// Mitsubishi GX Works2 project: Q-123_E_MTL   PLC: Q06H
// MDAS sample program

PROGRAM Q  // MDAS
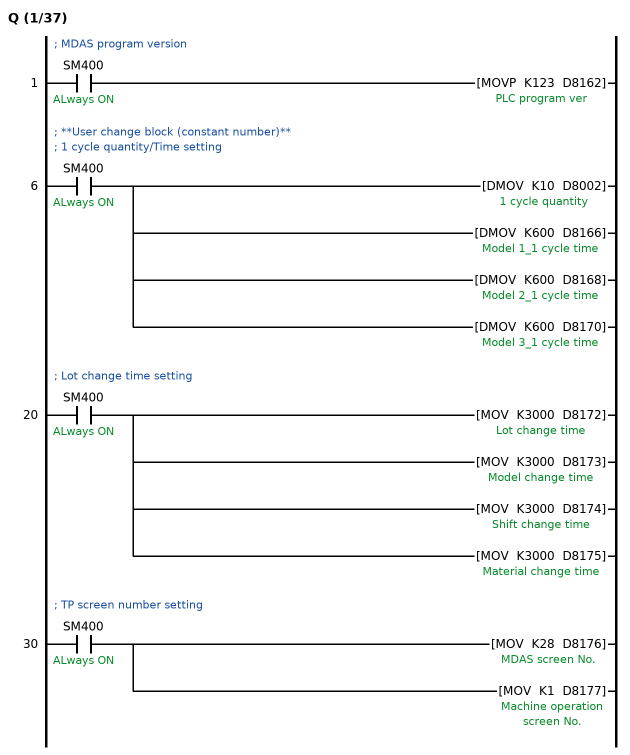
; MDAS program version
1     LD      SM400  ; ALways ON
      MOVP    K123 D8162  ; PLC program ver
; **User change block (constant number)**
; 1 cycle quantity/Time setting
6     LD      SM400  ; ALways ON
      DMOV    K10 D8002  ; 1 cycle quantity
      DMOV    K600 D8166  ; Model 1_1 cycle time
      DMOV    K600 D8168  ; Model 2_1 cycle time
      DMOV    K600 D8170  ; Model 3_1 cycle time
; Lot change time setting
20    LD      SM400  ; ALways ON
      MOV     K3000 D8172  ; Lot change time
      MOV     K3000 D8173  ; Model change time
      MOV     K3000 D8174  ; Shift change time
      MOV     K3000 D8175  ; Material change time
; TP screen number setting
30    LD      SM400  ; ALways ON
      MOV     K28 D8176  ; MDAS screen No.
      MOV     K1 D8177  ; Machine operation screen No.
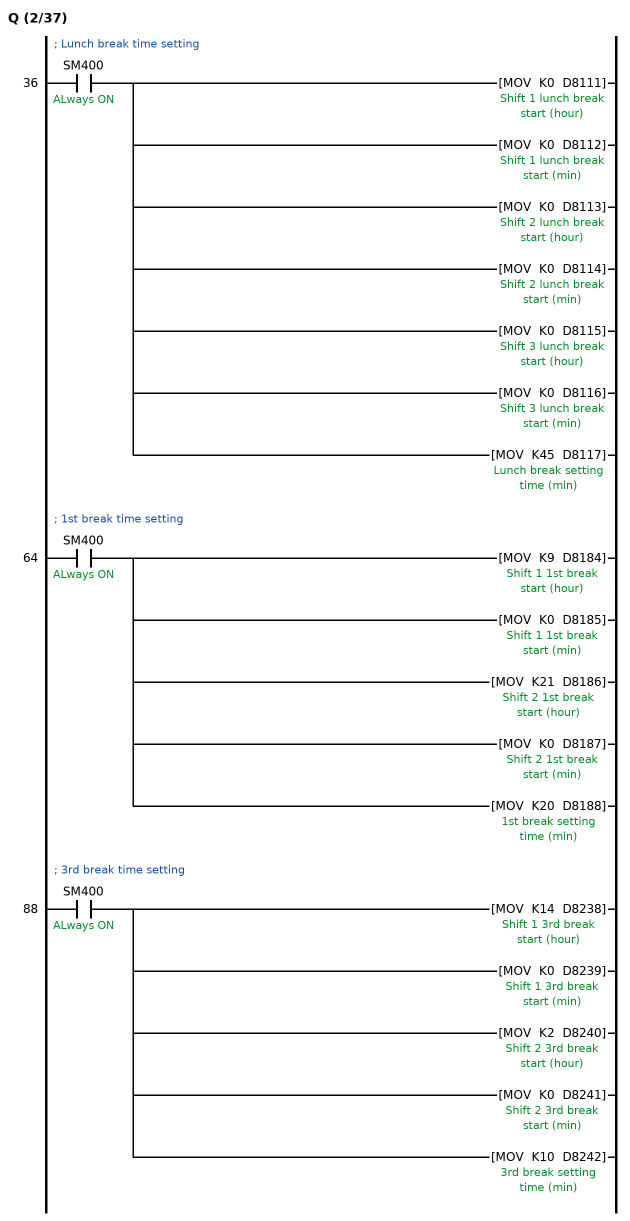
; Lunch break time setting
36    LD      SM400  ; ALways ON
      MOV     K0 D8111  ; Shift 1 lunch break start (hour)
      MOV     K0 D8112  ; Shift 1 lunch break start (min)
      MOV     K0 D8113  ; Shift 2 lunch break start (hour)
      MOV     K0 D8114  ; Shift 2 lunch break start (min)
      MOV     K0 D8115  ; Shift 3 lunch break start (hour)
      MOV     K0 D8116  ; Shift 3 lunch break start (min)
      MOV     K45 D8117  ; Lunch break setting time (min)
; 1st break time setting
64    LD      SM400  ; ALways ON
      MOV     K9 D8184  ; Shift 1 1st break start (hour)
      MOV     K0 D8185  ; Shift 1 1st break start (min)
      MOV     K21 D8186  ; Shift 2 1st break start (hour)
      MOV     K0 D8187  ; Shift 2 1st break start (min)
      MOV     K20 D8188  ; 1st break setting time (min)
; 3rd break time setting
88    LD      SM400  ; ALways ON
      MOV     K14 D8238  ; Shift 1 3rd break start (hour)
      MOV     K0 D8239  ; Shift 1 3rd break start (min)
      MOV     K2 D8240  ; Shift 2 3rd break start (hour)
      MOV     K0 D8241  ; Shift 2 3rd break start (min)
      MOV     K10 D8242  ; 3rd break setting time (min)
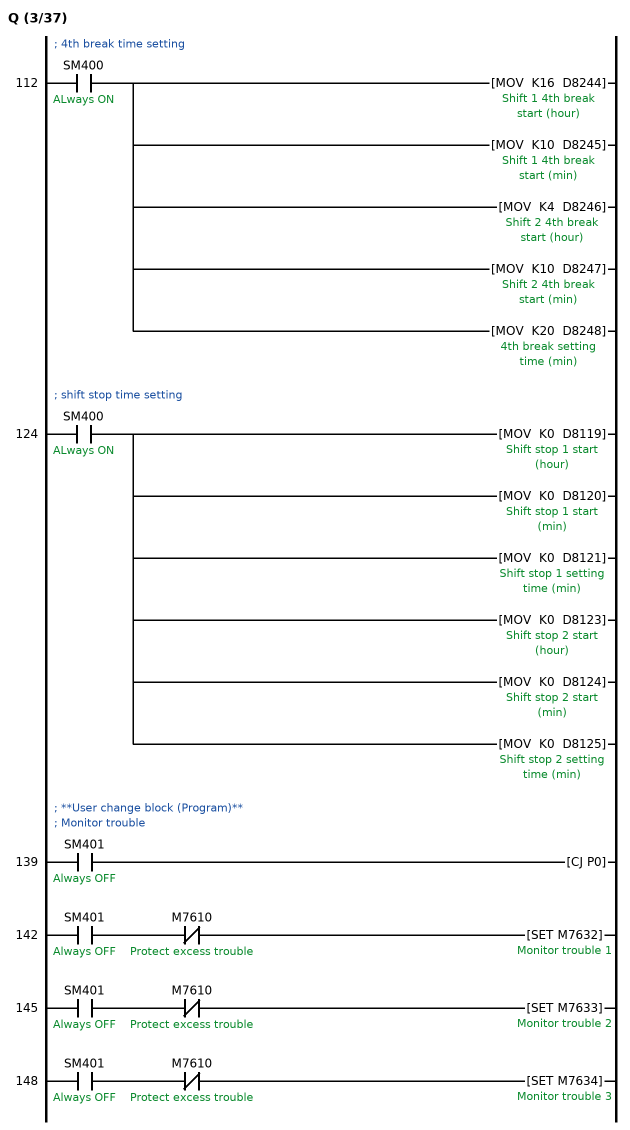
; 4th break time setting
112   LD      SM400  ; ALways ON
      MOV     K16 D8244  ; Shift 1 4th break start (hour)
      MOV     K10 D8245  ; Shift 1 4th break start (min)
      MOV     K4 D8246  ; Shift 2 4th break start (hour)
      MOV     K10 D8247  ; Shift 2 4th break start (min)
      MOV     K20 D8248  ; 4th break setting time (min)
; shift stop time setting
124   LD      SM400  ; ALways ON
      MOV     K0 D8119  ; Shift stop 1 start (hour)
      MOV     K0 D8120  ; Shift stop 1 start (min)
      MOV     K0 D8121  ; Shift stop 1 setting time (min)
      MOV     K0 D8123  ; Shift stop 2 start (hour)
      MOV     K0 D8124  ; Shift stop 2 start (min)
      MOV     K0 D8125  ; Shift stop 2 setting time (min)
; **User change block (Program)**
; Monitor trouble
139   LD      SM401  ; Always OFF
      CJ      P0
142   LD      SM401  ; Always OFF
      ANI     M7610  ; Protect excess trouble
      SET     M7632  ; Monitor trouble 1
145   LD      SM401  ; Always OFF
      ANI     M7610  ; Protect excess trouble
      SET     M7633  ; Monitor trouble 2
148   LD      SM401  ; Always OFF
      ANI     M7610  ; Protect excess trouble
      SET     M7634  ; Monitor trouble 3
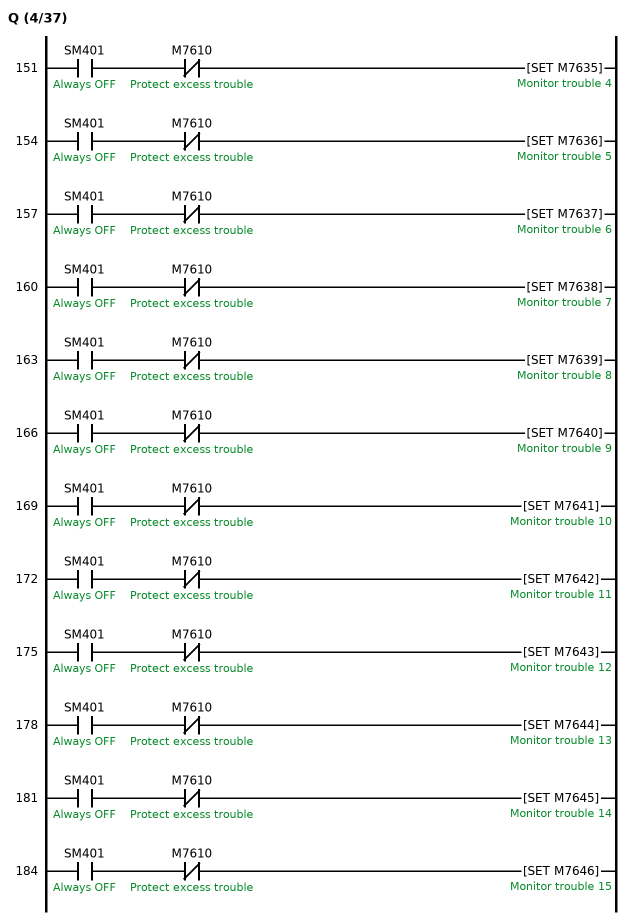
151   LD      SM401  ; Always OFF
      ANI     M7610  ; Protect excess trouble
      SET     M7635  ; Monitor trouble 4
154   LD      SM401  ; Always OFF
      ANI     M7610  ; Protect excess trouble
      SET     M7636  ; Monitor trouble 5
157   LD      SM401  ; Always OFF
      ANI     M7610  ; Protect excess trouble
      SET     M7637  ; Monitor trouble 6
160   LD      SM401  ; Always OFF
      ANI     M7610  ; Protect excess trouble
      SET     M7638  ; Monitor trouble 7
163   LD      SM401  ; Always OFF
      ANI     M7610  ; Protect excess trouble
      SET     M7639  ; Monitor trouble 8
166   LD      SM401  ; Always OFF
      ANI     M7610  ; Protect excess trouble
      SET     M7640  ; Monitor trouble 9
169   LD      SM401  ; Always OFF
      ANI     M7610  ; Protect excess trouble
      SET     M7641  ; Monitor trouble 10
172   LD      SM401  ; Always OFF
      ANI     M7610  ; Protect excess trouble
      SET     M7642  ; Monitor trouble 11
175   LD      SM401  ; Always OFF
      ANI     M7610  ; Protect excess trouble
      SET     M7643  ; Monitor trouble 12
178   LD      SM401  ; Always OFF
      ANI     M7610  ; Protect excess trouble
      SET     M7644  ; Monitor trouble 13
181   LD      SM401  ; Always OFF
      ANI     M7610  ; Protect excess trouble
      SET     M7645  ; Monitor trouble 14
184   LD      SM401  ; Always OFF
      ANI     M7610  ; Protect excess trouble
      SET     M7646  ; Monitor trouble 15
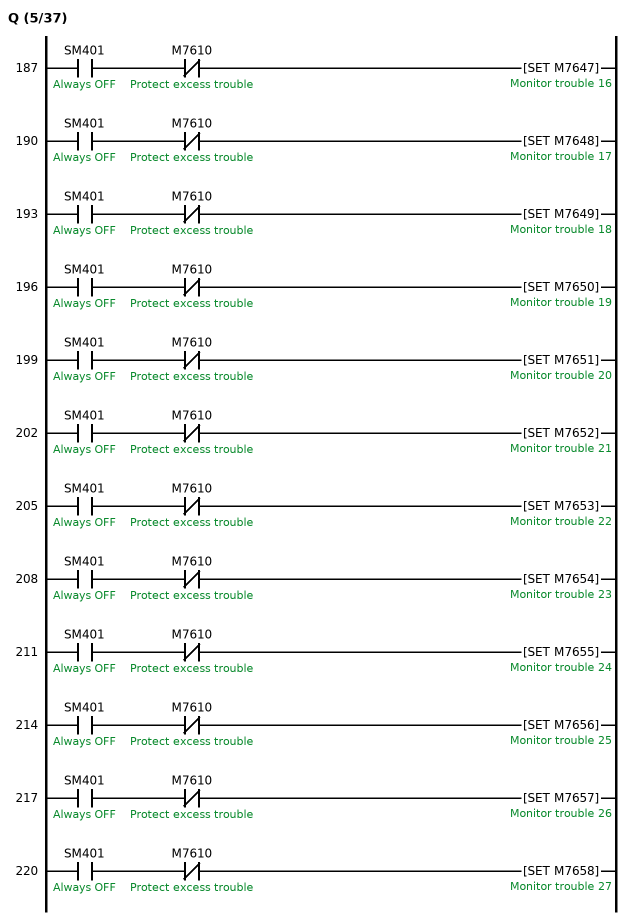
187   LD      SM401  ; Always OFF
      ANI     M7610  ; Protect excess trouble
      SET     M7647  ; Monitor trouble 16
190   LD      SM401  ; Always OFF
      ANI     M7610  ; Protect excess trouble
      SET     M7648  ; Monitor trouble 17
193   LD      SM401  ; Always OFF
      ANI     M7610  ; Protect excess trouble
      SET     M7649  ; Monitor trouble 18
196   LD      SM401  ; Always OFF
      ANI     M7610  ; Protect excess trouble
      SET     M7650  ; Monitor trouble 19
199   LD      SM401  ; Always OFF
      ANI     M7610  ; Protect excess trouble
      SET     M7651  ; Monitor trouble 20
202   LD      SM401  ; Always OFF
      ANI     M7610  ; Protect excess trouble
      SET     M7652  ; Monitor trouble 21
205   LD      SM401  ; Always OFF
      ANI     M7610  ; Protect excess trouble
      SET     M7653  ; Monitor trouble 22
208   LD      SM401  ; Always OFF
      ANI     M7610  ; Protect excess trouble
      SET     M7654  ; Monitor trouble 23
211   LD      SM401  ; Always OFF
      ANI     M7610  ; Protect excess trouble
      SET     M7655  ; Monitor trouble 24
214   LD      SM401  ; Always OFF
      ANI     M7610  ; Protect excess trouble
      SET     M7656  ; Monitor trouble 25
217   LD      SM401  ; Always OFF
      ANI     M7610  ; Protect excess trouble
      SET     M7657  ; Monitor trouble 26
220   LD      SM401  ; Always OFF
      ANI     M7610  ; Protect excess trouble
      SET     M7658  ; Monitor trouble 27
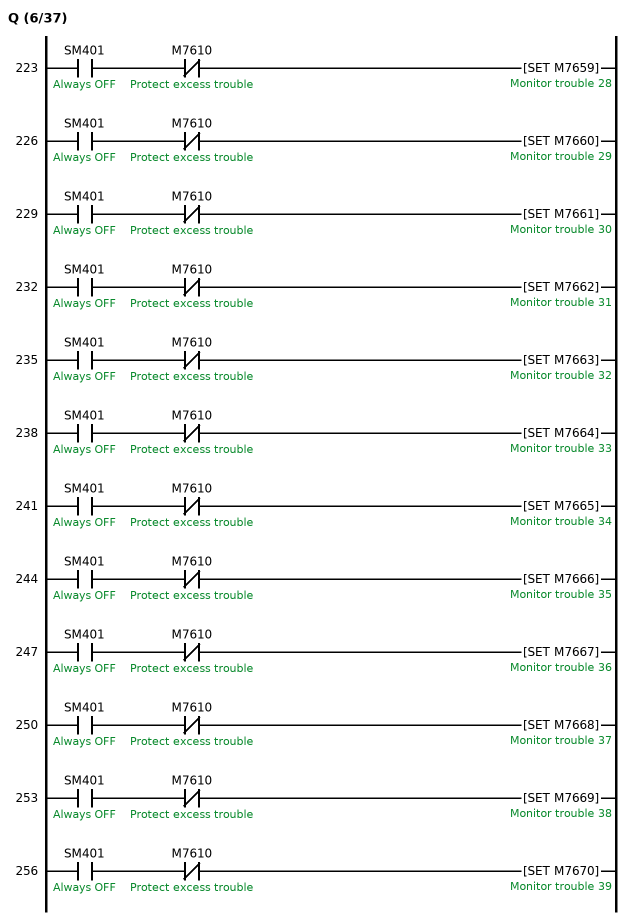
223   LD      SM401  ; Always OFF
      ANI     M7610  ; Protect excess trouble
      SET     M7659  ; Monitor trouble 28
226   LD      SM401  ; Always OFF
      ANI     M7610  ; Protect excess trouble
      SET     M7660  ; Monitor trouble 29
229   LD      SM401  ; Always OFF
      ANI     M7610  ; Protect excess trouble
      SET     M7661  ; Monitor trouble 30
232   LD      SM401  ; Always OFF
      ANI     M7610  ; Protect excess trouble
      SET     M7662  ; Monitor trouble 31
235   LD      SM401  ; Always OFF
      ANI     M7610  ; Protect excess trouble
      SET     M7663  ; Monitor trouble 32
238   LD      SM401  ; Always OFF
      ANI     M7610  ; Protect excess trouble
      SET     M7664  ; Monitor trouble 33
241   LD      SM401  ; Always OFF
      ANI     M7610  ; Protect excess trouble
      SET     M7665  ; Monitor trouble 34
244   LD      SM401  ; Always OFF
      ANI     M7610  ; Protect excess trouble
      SET     M7666  ; Monitor trouble 35
247   LD      SM401  ; Always OFF
      ANI     M7610  ; Protect excess trouble
      SET     M7667  ; Monitor trouble 36
250   LD      SM401  ; Always OFF
      ANI     M7610  ; Protect excess trouble
      SET     M7668  ; Monitor trouble 37
253   LD      SM401  ; Always OFF
      ANI     M7610  ; Protect excess trouble
      SET     M7669  ; Monitor trouble 38
256   LD      SM401  ; Always OFF
      ANI     M7610  ; Protect excess trouble
      SET     M7670  ; Monitor trouble 39
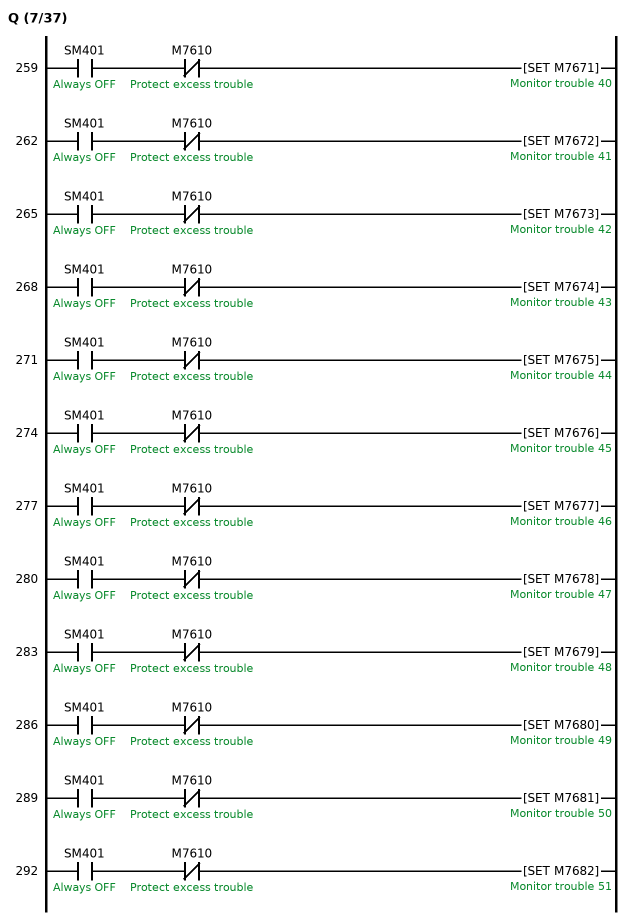
259   LD      SM401  ; Always OFF
      ANI     M7610  ; Protect excess trouble
      SET     M7671  ; Monitor trouble 40
262   LD      SM401  ; Always OFF
      ANI     M7610  ; Protect excess trouble
      SET     M7672  ; Monitor trouble 41
265   LD      SM401  ; Always OFF
      ANI     M7610  ; Protect excess trouble
      SET     M7673  ; Monitor trouble 42
268   LD      SM401  ; Always OFF
      ANI     M7610  ; Protect excess trouble
      SET     M7674  ; Monitor trouble 43
271   LD      SM401  ; Always OFF
      ANI     M7610  ; Protect excess trouble
      SET     M7675  ; Monitor trouble 44
274   LD      SM401  ; Always OFF
      ANI     M7610  ; Protect excess trouble
      SET     M7676  ; Monitor trouble 45
277   LD      SM401  ; Always OFF
      ANI     M7610  ; Protect excess trouble
      SET     M7677  ; Monitor trouble 46
280   LD      SM401  ; Always OFF
      ANI     M7610  ; Protect excess trouble
      SET     M7678  ; Monitor trouble 47
283   LD      SM401  ; Always OFF
      ANI     M7610  ; Protect excess trouble
      SET     M7679  ; Monitor trouble 48
286   LD      SM401  ; Always OFF
      ANI     M7610  ; Protect excess trouble
      SET     M7680  ; Monitor trouble 49
289   LD      SM401  ; Always OFF
      ANI     M7610  ; Protect excess trouble
      SET     M7681  ; Monitor trouble 50
292   LD      SM401  ; Always OFF
      ANI     M7610  ; Protect excess trouble
      SET     M7682  ; Monitor trouble 51
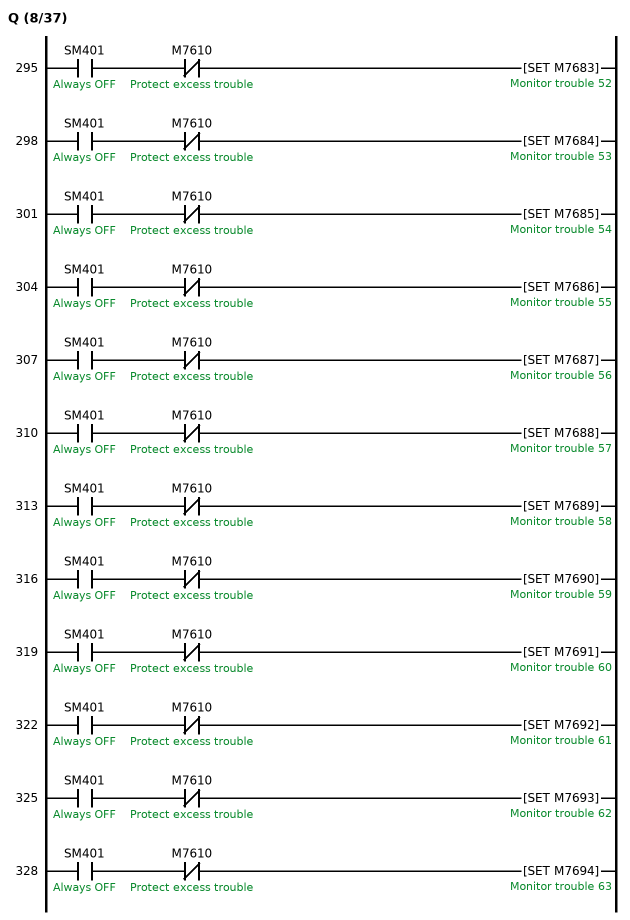
295   LD      SM401  ; Always OFF
      ANI     M7610  ; Protect excess trouble
      SET     M7683  ; Monitor trouble 52
298   LD      SM401  ; Always OFF
      ANI     M7610  ; Protect excess trouble
      SET     M7684  ; Monitor trouble 53
301   LD      SM401  ; Always OFF
      ANI     M7610  ; Protect excess trouble
      SET     M7685  ; Monitor trouble 54
304   LD      SM401  ; Always OFF
      ANI     M7610  ; Protect excess trouble
      SET     M7686  ; Monitor trouble 55
307   LD      SM401  ; Always OFF
      ANI     M7610  ; Protect excess trouble
      SET     M7687  ; Monitor trouble 56
310   LD      SM401  ; Always OFF
      ANI     M7610  ; Protect excess trouble
      SET     M7688  ; Monitor trouble 57
313   LD      SM401  ; Always OFF
      ANI     M7610  ; Protect excess trouble
      SET     M7689  ; Monitor trouble 58
316   LD      SM401  ; Always OFF
      ANI     M7610  ; Protect excess trouble
      SET     M7690  ; Monitor trouble 59
319   LD      SM401  ; Always OFF
      ANI     M7610  ; Protect excess trouble
      SET     M7691  ; Monitor trouble 60
322   LD      SM401  ; Always OFF
      ANI     M7610  ; Protect excess trouble
      SET     M7692  ; Monitor trouble 61
325   LD      SM401  ; Always OFF
      ANI     M7610  ; Protect excess trouble
      SET     M7693  ; Monitor trouble 62
328   LD      SM401  ; Always OFF
      ANI     M7610  ; Protect excess trouble
      SET     M7694  ; Monitor trouble 63
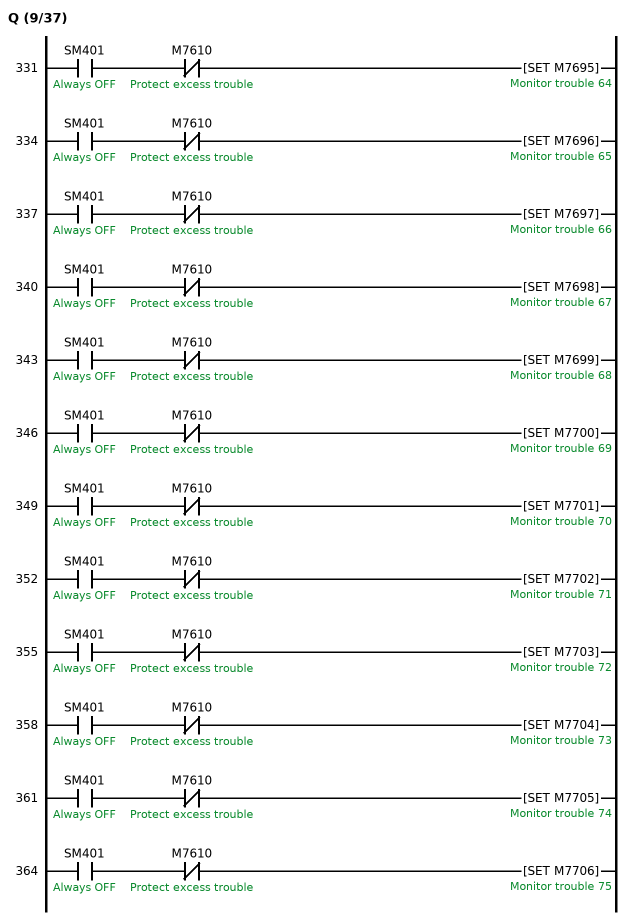
331   LD      SM401  ; Always OFF
      ANI     M7610  ; Protect excess trouble
      SET     M7695  ; Monitor trouble 64
334   LD      SM401  ; Always OFF
      ANI     M7610  ; Protect excess trouble
      SET     M7696  ; Monitor trouble 65
337   LD      SM401  ; Always OFF
      ANI     M7610  ; Protect excess trouble
      SET     M7697  ; Monitor trouble 66
340   LD      SM401  ; Always OFF
      ANI     M7610  ; Protect excess trouble
      SET     M7698  ; Monitor trouble 67
343   LD      SM401  ; Always OFF
      ANI     M7610  ; Protect excess trouble
      SET     M7699  ; Monitor trouble 68
346   LD      SM401  ; Always OFF
      ANI     M7610  ; Protect excess trouble
      SET     M7700  ; Monitor trouble 69
349   LD      SM401  ; Always OFF
      ANI     M7610  ; Protect excess trouble
      SET     M7701  ; Monitor trouble 70
352   LD      SM401  ; Always OFF
      ANI     M7610  ; Protect excess trouble
      SET     M7702  ; Monitor trouble 71
355   LD      SM401  ; Always OFF
      ANI     M7610  ; Protect excess trouble
      SET     M7703  ; Monitor trouble 72
358   LD      SM401  ; Always OFF
      ANI     M7610  ; Protect excess trouble
      SET     M7704  ; Monitor trouble 73
361   LD      SM401  ; Always OFF
      ANI     M7610  ; Protect excess trouble
      SET     M7705  ; Monitor trouble 74
364   LD      SM401  ; Always OFF
      ANI     M7610  ; Protect excess trouble
      SET     M7706  ; Monitor trouble 75
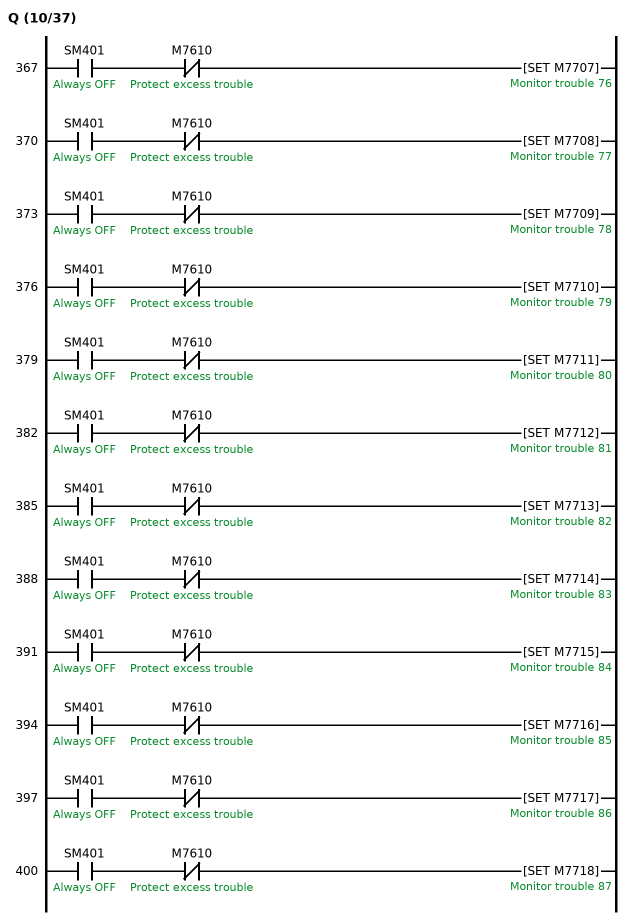
367   LD      SM401  ; Always OFF
      ANI     M7610  ; Protect excess trouble
      SET     M7707  ; Monitor trouble 76
370   LD      SM401  ; Always OFF
      ANI     M7610  ; Protect excess trouble
      SET     M7708  ; Monitor trouble 77
373   LD      SM401  ; Always OFF
      ANI     M7610  ; Protect excess trouble
      SET     M7709  ; Monitor trouble 78
376   LD      SM401  ; Always OFF
      ANI     M7610  ; Protect excess trouble
      SET     M7710  ; Monitor trouble 79
379   LD      SM401  ; Always OFF
      ANI     M7610  ; Protect excess trouble
      SET     M7711  ; Monitor trouble 80
382   LD      SM401  ; Always OFF
      ANI     M7610  ; Protect excess trouble
      SET     M7712  ; Monitor trouble 81
385   LD      SM401  ; Always OFF
      ANI     M7610  ; Protect excess trouble
      SET     M7713  ; Monitor trouble 82
388   LD      SM401  ; Always OFF
      ANI     M7610  ; Protect excess trouble
      SET     M7714  ; Monitor trouble 83
391   LD      SM401  ; Always OFF
      ANI     M7610  ; Protect excess trouble
      SET     M7715  ; Monitor trouble 84
394   LD      SM401  ; Always OFF
      ANI     M7610  ; Protect excess trouble
      SET     M7716  ; Monitor trouble 85
397   LD      SM401  ; Always OFF
      ANI     M7610  ; Protect excess trouble
      SET     M7717  ; Monitor trouble 86
400   LD      SM401  ; Always OFF
      ANI     M7610  ; Protect excess trouble
      SET     M7718  ; Monitor trouble 87
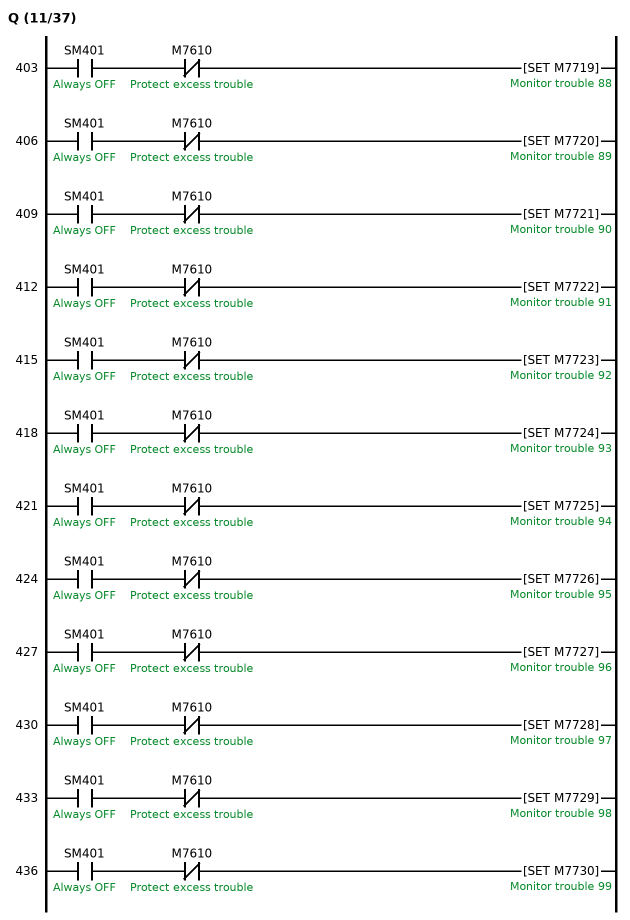
403   LD      SM401  ; Always OFF
      ANI     M7610  ; Protect excess trouble
      SET     M7719  ; Monitor trouble 88
406   LD      SM401  ; Always OFF
      ANI     M7610  ; Protect excess trouble
      SET     M7720  ; Monitor trouble 89
409   LD      SM401  ; Always OFF
      ANI     M7610  ; Protect excess trouble
      SET     M7721  ; Monitor trouble 90
412   LD      SM401  ; Always OFF
      ANI     M7610  ; Protect excess trouble
      SET     M7722  ; Monitor trouble 91
415   LD      SM401  ; Always OFF
      ANI     M7610  ; Protect excess trouble
      SET     M7723  ; Monitor trouble 92
418   LD      SM401  ; Always OFF
      ANI     M7610  ; Protect excess trouble
      SET     M7724  ; Monitor trouble 93
421   LD      SM401  ; Always OFF
      ANI     M7610  ; Protect excess trouble
      SET     M7725  ; Monitor trouble 94
424   LD      SM401  ; Always OFF
      ANI     M7610  ; Protect excess trouble
      SET     M7726  ; Monitor trouble 95
427   LD      SM401  ; Always OFF
      ANI     M7610  ; Protect excess trouble
      SET     M7727  ; Monitor trouble 96
430   LD      SM401  ; Always OFF
      ANI     M7610  ; Protect excess trouble
      SET     M7728  ; Monitor trouble 97
433   LD      SM401  ; Always OFF
      ANI     M7610  ; Protect excess trouble
      SET     M7729  ; Monitor trouble 98
436   LD      SM401  ; Always OFF
      ANI     M7610  ; Protect excess trouble
      SET     M7730  ; Monitor trouble 99
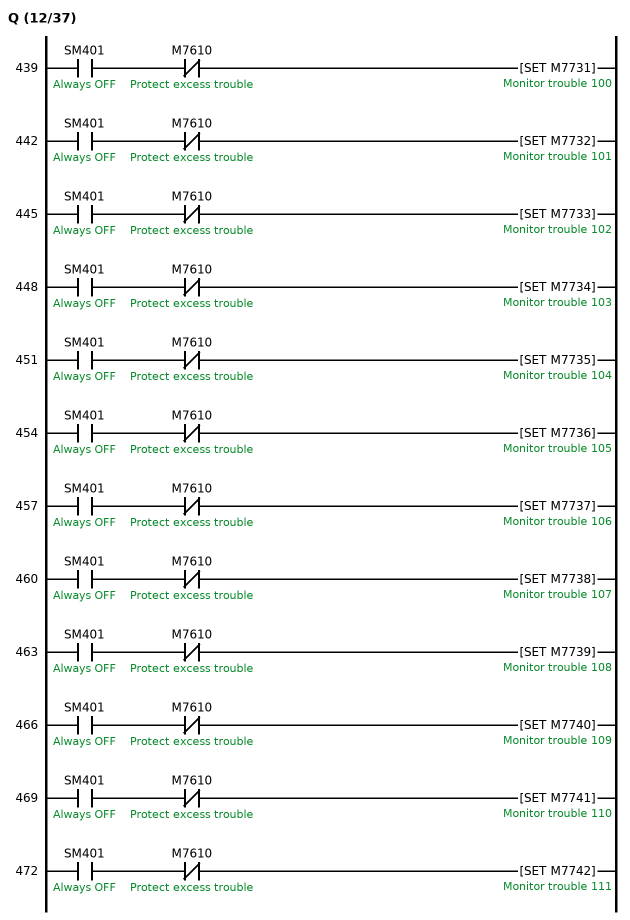
439   LD      SM401  ; Always OFF
      ANI     M7610  ; Protect excess trouble
      SET     M7731  ; Monitor trouble 100
442   LD      SM401  ; Always OFF
      ANI     M7610  ; Protect excess trouble
      SET     M7732  ; Monitor trouble 101
445   LD      SM401  ; Always OFF
      ANI     M7610  ; Protect excess trouble
      SET     M7733  ; Monitor trouble 102
448   LD      SM401  ; Always OFF
      ANI     M7610  ; Protect excess trouble
      SET     M7734  ; Monitor trouble 103
451   LD      SM401  ; Always OFF
      ANI     M7610  ; Protect excess trouble
      SET     M7735  ; Monitor trouble 104
454   LD      SM401  ; Always OFF
      ANI     M7610  ; Protect excess trouble
      SET     M7736  ; Monitor trouble 105
457   LD      SM401  ; Always OFF
      ANI     M7610  ; Protect excess trouble
      SET     M7737  ; Monitor trouble 106
460   LD      SM401  ; Always OFF
      ANI     M7610  ; Protect excess trouble
      SET     M7738  ; Monitor trouble 107
463   LD      SM401  ; Always OFF
      ANI     M7610  ; Protect excess trouble
      SET     M7739  ; Monitor trouble 108
466   LD      SM401  ; Always OFF
      ANI     M7610  ; Protect excess trouble
      SET     M7740  ; Monitor trouble 109
469   LD      SM401  ; Always OFF
      ANI     M7610  ; Protect excess trouble
      SET     M7741  ; Monitor trouble 110
472   LD      SM401  ; Always OFF
      ANI     M7610  ; Protect excess trouble
      SET     M7742  ; Monitor trouble 111
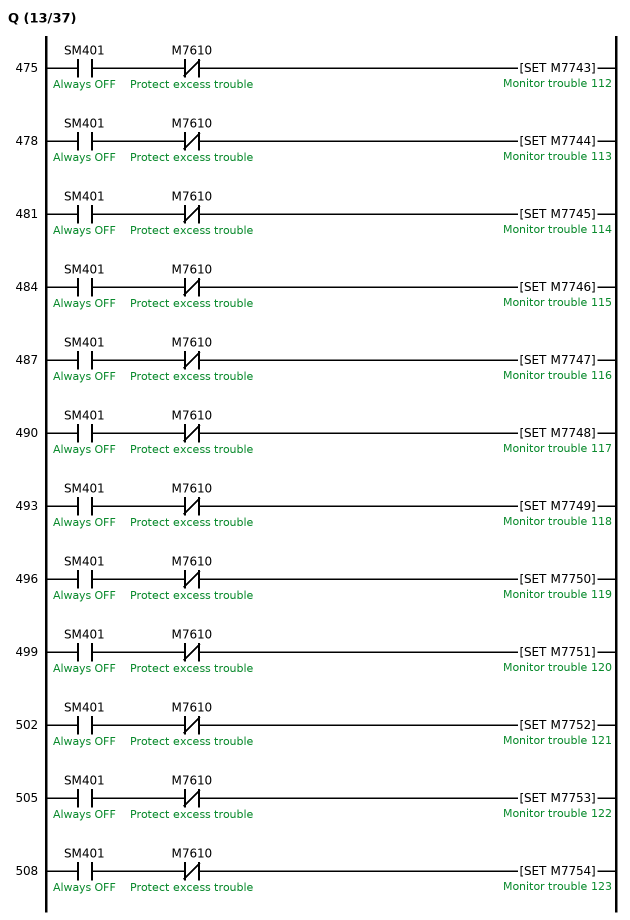
475   LD      SM401  ; Always OFF
      ANI     M7610  ; Protect excess trouble
      SET     M7743  ; Monitor trouble 112
478   LD      SM401  ; Always OFF
      ANI     M7610  ; Protect excess trouble
      SET     M7744  ; Monitor trouble 113
481   LD      SM401  ; Always OFF
      ANI     M7610  ; Protect excess trouble
      SET     M7745  ; Monitor trouble 114
484   LD      SM401  ; Always OFF
      ANI     M7610  ; Protect excess trouble
      SET     M7746  ; Monitor trouble 115
487   LD      SM401  ; Always OFF
      ANI     M7610  ; Protect excess trouble
      SET     M7747  ; Monitor trouble 116
490   LD      SM401  ; Always OFF
      ANI     M7610  ; Protect excess trouble
      SET     M7748  ; Monitor trouble 117
493   LD      SM401  ; Always OFF
      ANI     M7610  ; Protect excess trouble
      SET     M7749  ; Monitor trouble 118
496   LD      SM401  ; Always OFF
      ANI     M7610  ; Protect excess trouble
      SET     M7750  ; Monitor trouble 119
499   LD      SM401  ; Always OFF
      ANI     M7610  ; Protect excess trouble
      SET     M7751  ; Monitor trouble 120
502   LD      SM401  ; Always OFF
      ANI     M7610  ; Protect excess trouble
      SET     M7752  ; Monitor trouble 121
505   LD      SM401  ; Always OFF
      ANI     M7610  ; Protect excess trouble
      SET     M7753  ; Monitor trouble 122
508   LD      SM401  ; Always OFF
      ANI     M7610  ; Protect excess trouble
      SET     M7754  ; Monitor trouble 123
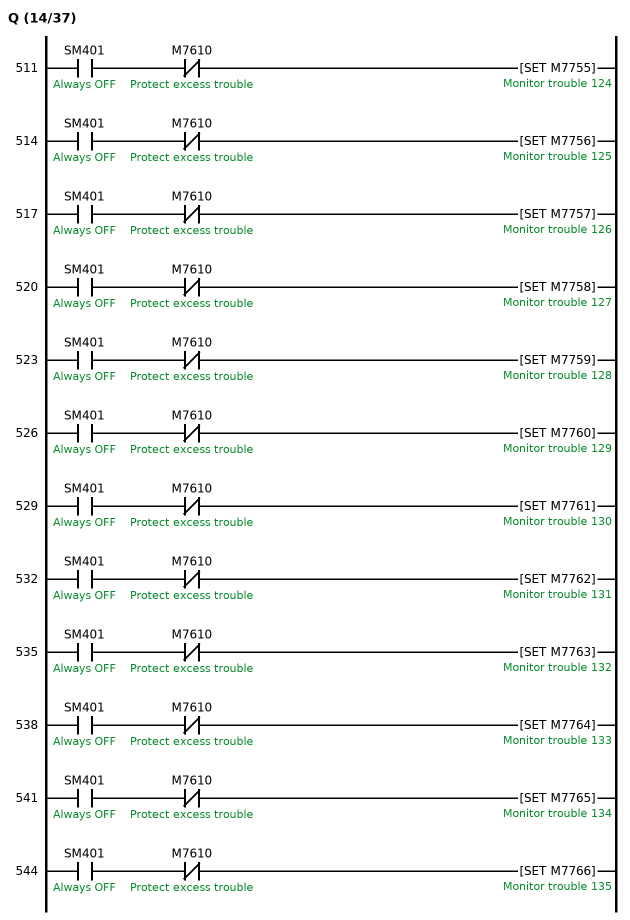
511   LD      SM401  ; Always OFF
      ANI     M7610  ; Protect excess trouble
      SET     M7755  ; Monitor trouble 124
514   LD      SM401  ; Always OFF
      ANI     M7610  ; Protect excess trouble
      SET     M7756  ; Monitor trouble 125
517   LD      SM401  ; Always OFF
      ANI     M7610  ; Protect excess trouble
      SET     M7757  ; Monitor trouble 126
520   LD      SM401  ; Always OFF
      ANI     M7610  ; Protect excess trouble
      SET     M7758  ; Monitor trouble 127
523   LD      SM401  ; Always OFF
      ANI     M7610  ; Protect excess trouble
      SET     M7759  ; Monitor trouble 128
526   LD      SM401  ; Always OFF
      ANI     M7610  ; Protect excess trouble
      SET     M7760  ; Monitor trouble 129
529   LD      SM401  ; Always OFF
      ANI     M7610  ; Protect excess trouble
      SET     M7761  ; Monitor trouble 130
532   LD      SM401  ; Always OFF
      ANI     M7610  ; Protect excess trouble
      SET     M7762  ; Monitor trouble 131
535   LD      SM401  ; Always OFF
      ANI     M7610  ; Protect excess trouble
      SET     M7763  ; Monitor trouble 132
538   LD      SM401  ; Always OFF
      ANI     M7610  ; Protect excess trouble
      SET     M7764  ; Monitor trouble 133
541   LD      SM401  ; Always OFF
      ANI     M7610  ; Protect excess trouble
      SET     M7765  ; Monitor trouble 134
544   LD      SM401  ; Always OFF
      ANI     M7610  ; Protect excess trouble
      SET     M7766  ; Monitor trouble 135
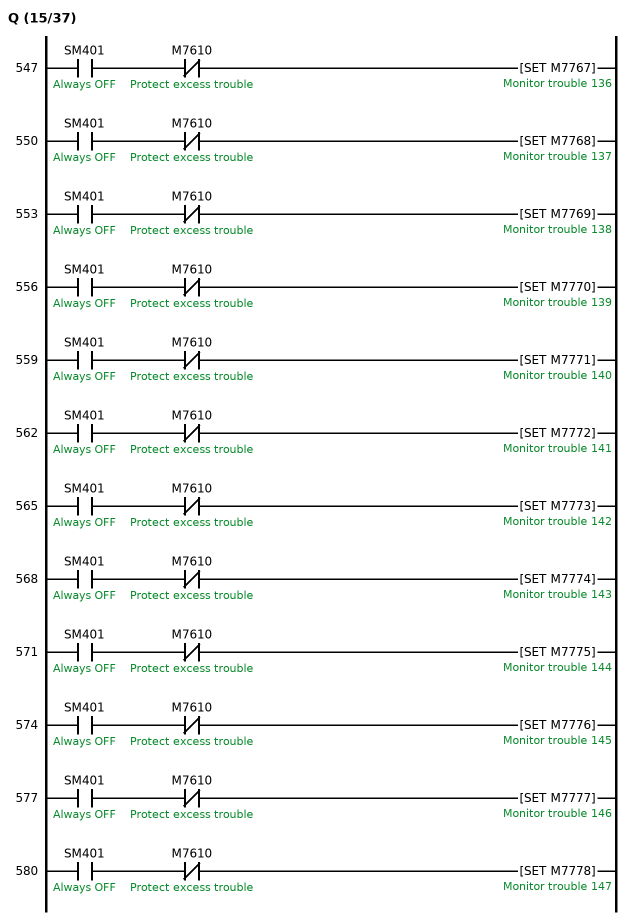
547   LD      SM401  ; Always OFF
      ANI     M7610  ; Protect excess trouble
      SET     M7767  ; Monitor trouble 136
550   LD      SM401  ; Always OFF
      ANI     M7610  ; Protect excess trouble
      SET     M7768  ; Monitor trouble 137
553   LD      SM401  ; Always OFF
      ANI     M7610  ; Protect excess trouble
      SET     M7769  ; Monitor trouble 138
556   LD      SM401  ; Always OFF
      ANI     M7610  ; Protect excess trouble
      SET     M7770  ; Monitor trouble 139
559   LD      SM401  ; Always OFF
      ANI     M7610  ; Protect excess trouble
      SET     M7771  ; Monitor trouble 140
562   LD      SM401  ; Always OFF
      ANI     M7610  ; Protect excess trouble
      SET     M7772  ; Monitor trouble 141
565   LD      SM401  ; Always OFF
      ANI     M7610  ; Protect excess trouble
      SET     M7773  ; Monitor trouble 142
568   LD      SM401  ; Always OFF
      ANI     M7610  ; Protect excess trouble
      SET     M7774  ; Monitor trouble 143
571   LD      SM401  ; Always OFF
      ANI     M7610  ; Protect excess trouble
      SET     M7775  ; Monitor trouble 144
574   LD      SM401  ; Always OFF
      ANI     M7610  ; Protect excess trouble
      SET     M7776  ; Monitor trouble 145
577   LD      SM401  ; Always OFF
      ANI     M7610  ; Protect excess trouble
      SET     M7777  ; Monitor trouble 146
580   LD      SM401  ; Always OFF
      ANI     M7610  ; Protect excess trouble
      SET     M7778  ; Monitor trouble 147
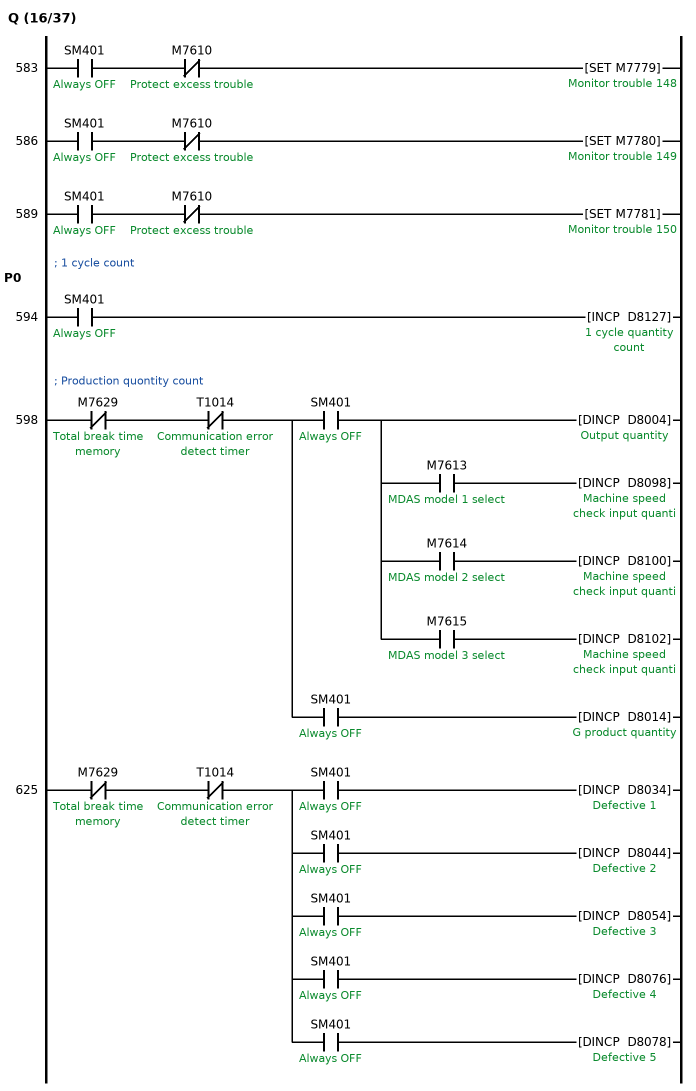
583   LD      SM401  ; Always OFF
      ANI     M7610  ; Protect excess trouble
      SET     M7779  ; Monitor trouble 148
586   LD      SM401  ; Always OFF
      ANI     M7610  ; Protect excess trouble
      SET     M7780  ; Monitor trouble 149
589   LD      SM401  ; Always OFF
      ANI     M7610  ; Protect excess trouble
      SET     M7781  ; Monitor trouble 150
; 1 cycle count
      P0
594   LD      SM401  ; Always OFF
      INCP    D8127  ; 1 cycle quantity count
; Production quontity count
598   LDI     M7629  ; Total break time memory
      ANI     T1014  ; Communication error detect timer
      MPS
      AND     SM401  ; Always OFF
      DINCP   D8004  ; Output quantity
      MPS
      AND     M7613  ; MDAS model 1 select
      DINCP   D8098  ; Machine speed check input quanti
      MRD
      AND     M7614  ; MDAS model 2 select
      DINCP   D8100  ; Machine speed check input quanti
      MPP
      AND     M7615  ; MDAS model 3 select
      DINCP   D8102  ; Machine speed check input quanti
      MPP
      AND     SM401  ; Always OFF
      DINCP   D8014  ; G product quantity
625   LDI     M7629  ; Total break time memory
      ANI     T1014  ; Communication error detect timer
      MPS
      AND     SM401  ; Always OFF
      DINCP   D8034  ; Defective 1
      MRD
      AND     SM401  ; Always OFF
      DINCP   D8044  ; Defective 2
      MRD
      AND     SM401  ; Always OFF
      DINCP   D8054  ; Defective 3
      MRD
      AND     SM401  ; Always OFF
      DINCP   D8076  ; Defective 4
      MPP
      AND     SM401  ; Always OFF
      DINCP   D8078  ; Defective 5
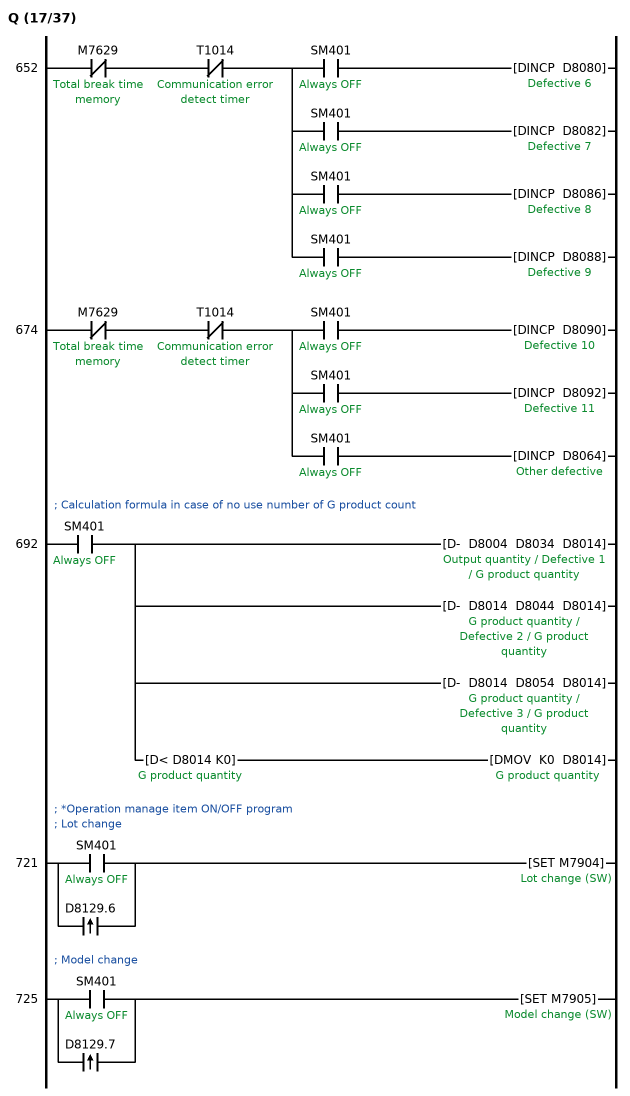
652   LDI     M7629  ; Total break time memory
      ANI     T1014  ; Communication error detect timer
      MPS
      AND     SM401  ; Always OFF
      DINCP   D8080  ; Defective 6
      MRD
      AND     SM401  ; Always OFF
      DINCP   D8082  ; Defective 7
      MRD
      AND     SM401  ; Always OFF
      DINCP   D8086  ; Defective 8
      MPP
      AND     SM401  ; Always OFF
      DINCP   D8088  ; Defective 9
674   LDI     M7629  ; Total break time memory
      ANI     T1014  ; Communication error detect timer
      MPS
      AND     SM401  ; Always OFF
      DINCP   D8090  ; Defective 10
      MRD
      AND     SM401  ; Always OFF
      DINCP   D8092  ; Defective 11
      MPP
      AND     SM401  ; Always OFF
      DINCP   D8064  ; Other defective
; Calculation formula in case of no use number of G product count
692   LD      SM401  ; Always OFF
      D-      D8004 D8034 D8014
      D-      D8014 D8044 D8014
      D-      D8014 D8054 D8014
      ANDD<   D8014 K0  ; G product quantity
      DMOV    K0 D8014
; *Operation manage item ON/OFF program
; Lot change
721   LD      SM401  ; Always OFF
      ORP     D8129.6
      SET     M7904  ; Lot change (SW)
; Model change
725   LD      SM401  ; Always OFF
      ORP     D8129.7
      SET     M7905  ; Model change (SW)
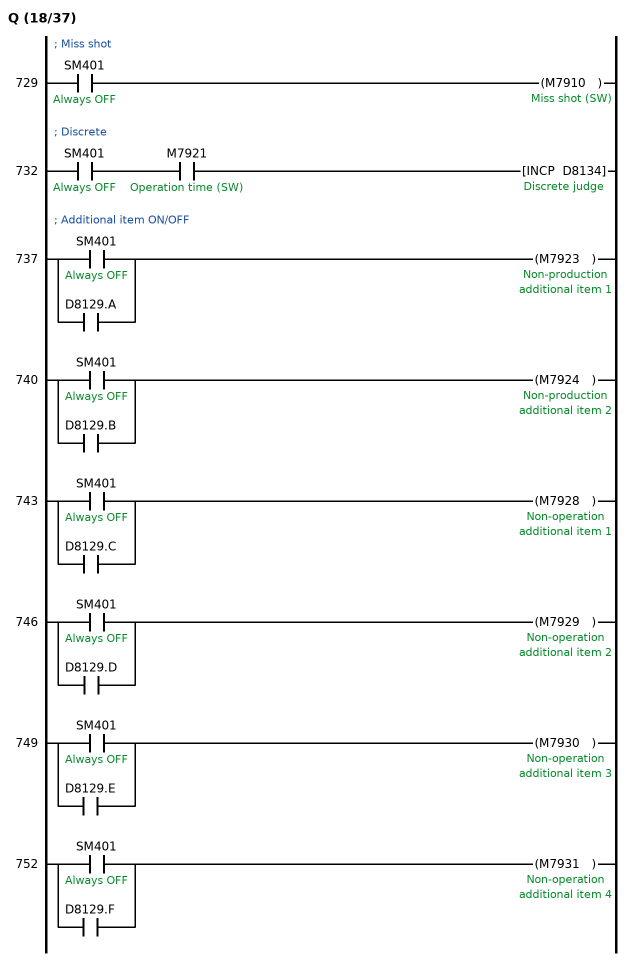
; Miss shot
729   LD      SM401  ; Always OFF
      OUT     M7910  ; Miss shot (SW)
; Discrete
732   LD      SM401  ; Always OFF
      AND     M7921  ; Operation time (SW)
      INCP    D8134  ; Discrete judge
; Additional item ON/OFF
737   LD      SM401  ; Always OFF
      OR      D8129.A
      OUT     M7923  ; Non-production additional item 1
740   LD      SM401  ; Always OFF
      OR      D8129.B
      OUT     M7924  ; Non-production additional item 2
743   LD      SM401  ; Always OFF
      OR      D8129.C
      OUT     M7928  ; Non-operation additional item 1
746   LD      SM401  ; Always OFF
      OR      D8129.D
      OUT     M7929  ; Non-operation additional item 2
749   LD      SM401  ; Always OFF
      OR      D8129.E
      OUT     M7930  ; Non-operation additional item 3
752   LD      SM401  ; Always OFF
      OR      D8129.F
      OUT     M7931  ; Non-operation additional item 4
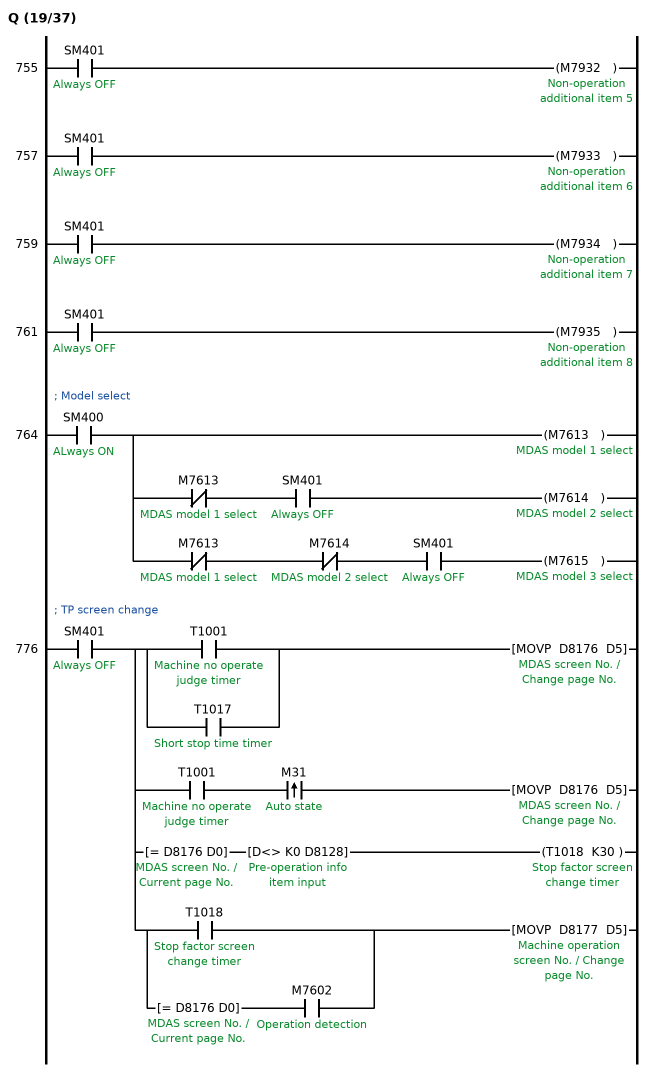
755   LD      SM401  ; Always OFF
      OUT     M7932  ; Non-operation additional item 5
757   LD      SM401  ; Always OFF
      OUT     M7933  ; Non-operation additional item 6
759   LD      SM401  ; Always OFF
      OUT     M7934  ; Non-operation additional item 7
761   LD      SM401  ; Always OFF
      OUT     M7935  ; Non-operation additional item 8
; Model select
764   LD      SM400  ; ALways ON
      OUT     M7613  ; MDAS model 1 select
      MPS
      ANI     M7613  ; MDAS model 1 select
      AND     SM401  ; Always OFF
      OUT     M7614  ; MDAS model 2 select
      MPP
      ANI     M7613  ; MDAS model 1 select
      ANI     M7614  ; MDAS model 2 select
      AND     SM401  ; Always OFF
      OUT     M7615  ; MDAS model 3 select
; TP screen change
776   LD      SM401  ; Always OFF
      MPS
      LD      T1001  ; Machine no operate judge timer
      OR      T1017  ; Short stop time timer
      ANB
      MOVP    D8176 D5  ; Change page No.
      MRD
      AND     T1001  ; Machine no operate judge timer
      ANDP    M31  ; Auto state
      MOVP    D8176 D5
      MRD
      AND=    D8176 D0  ; MDAS screen No. / Current page No.
      ANDD<>  K0 D8128  ; Pre-operation info item input
      OUT     T1018 K30  ; Stop factor screen change timer
      MPP
      LD      T1018  ; Stop factor screen change timer
      LD=     D8176 D0  ; MDAS screen No. / Current page No.
      AND     M7602  ; Operation detection
      ORB
      ANB
      MOVP    D8177 D5
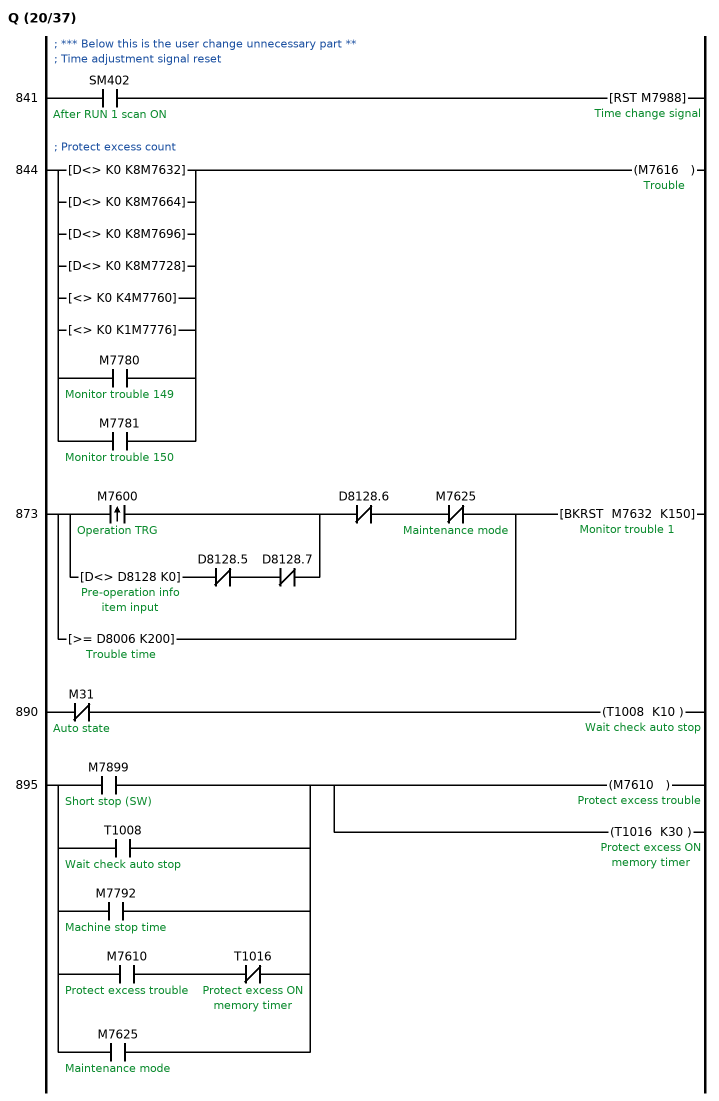
; *** Below this is the user change unnecessary part **
; Time adjustment signal reset
841   LD      SM402  ; After RUN 1 scan ON
      RST     M7988  ; Time change signal
; Protect excess count
844   LDD<>   K0 K8M7632  ; Monitor trouble 1
      ORD<>   K0 K8M7664  ; Monitor trouble 33
      ORD<>   K0 K8M7696  ; Monitor trouble 65
      ORD<>   K0 K8M7728  ; Monitor trouble 97
      OR<>    K0 K4M7760  ; Monitor trouble 129
      OR<>    K0 K1M7776  ; Monitor trouble 145
      OR      M7780  ; Monitor trouble 149
      OR      M7781  ; Monitor trouble 150
      OUT     M7616  ; Trouble
873   LDP     M7600  ; Operation TRG
      LDD<>   D8128 K0  ; Pre-operation info item input
      ANI     D8128.5
      ANI     D8128.7
      ORB
      ANI     D8128.6
      ANI     M7625  ; Maintenance mode
      OR>=    D8006 K200  ; Trouble time
      BKRST   M7632 K150
890   LDI     M31  ; Auto state
      OUT     T1008 K10  ; Wait check auto stop
895   LD      M7899  ; Short stop (SW)
      OR      T1008  ; Wait check auto stop
      OR      M7792  ; Machine stop time
      LD      M7610  ; Protect excess trouble
      ANI     T1016  ; Protect excess ON memory timer
      ORB
      OR      M7625  ; Maintenance mode
      OUT     M7610  ; Protect excess trouble
      OUT     T1016 K30  ; Protect excess ON memory timer
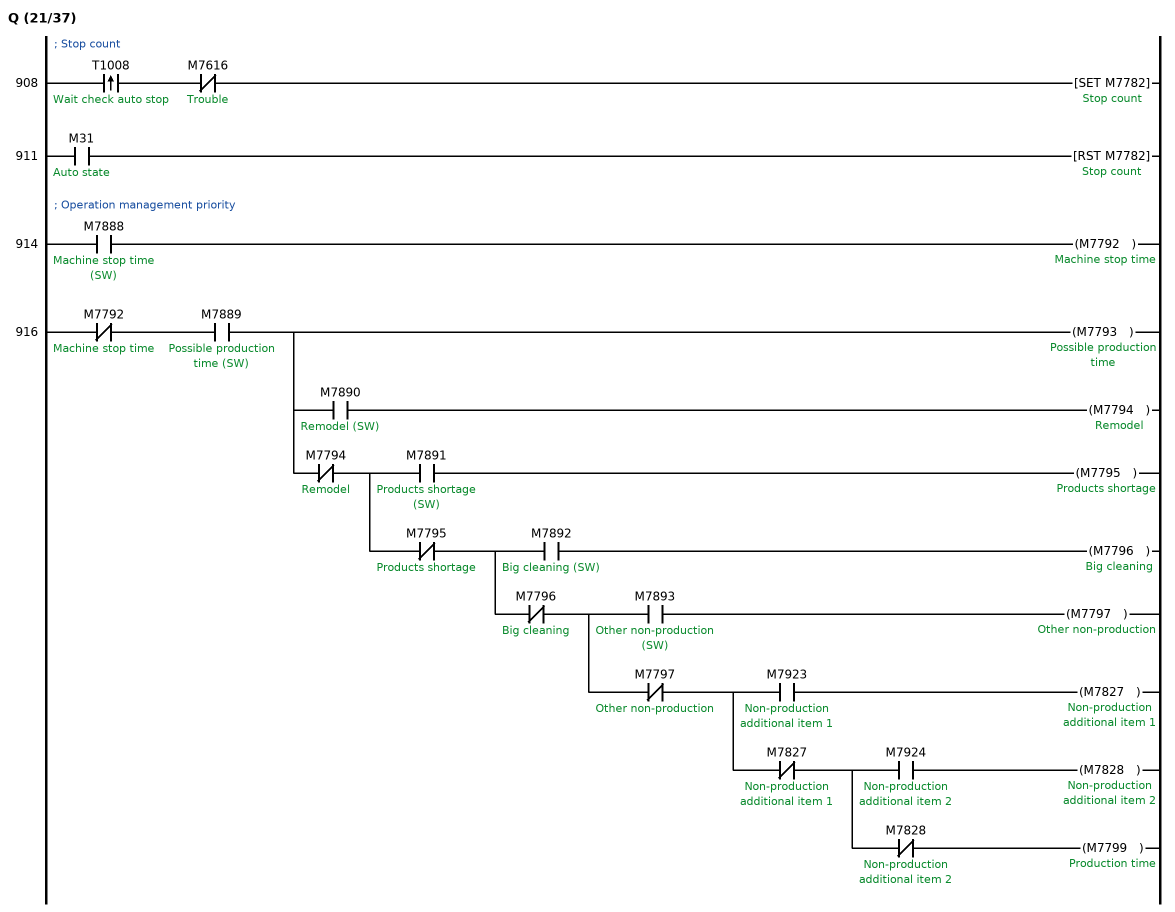
; Stop count
908   LDP     T1008  ; Wait check auto stop
      ANI     M7616  ; Trouble
      SET     M7782  ; Stop count
911   LD      M31  ; Auto state
      RST     M7782  ; Stop count
; Operation management priority
914   LD      M7888  ; Machine stop time (SW)
      OUT     M7792  ; Machine stop time
916   LDI     M7792  ; Machine stop time
      AND     M7889  ; Possible production time (SW)
      OUT     M7793  ; Possible production time
      MPS
      AND     M7890  ; Remodel (SW)
      OUT     M7794  ; Remodel
      MPP
      ANI     M7794  ; Remodel
      MPS
      AND     M7891  ; Products shortage (SW)
      OUT     M7795  ; Products shortage
      MPP
      ANI     M7795  ; Products shortage
      MPS
      AND     M7892  ; Big cleaning (SW)
      OUT     M7796  ; Big cleaning
      MPP
      ANI     M7796  ; Big cleaning
      MPS
      AND     M7893  ; Other non-production (SW)
      OUT     M7797  ; Other non-production
      MPP
      ANI     M7797  ; Other non-production
      MPS
      AND     M7923  ; Non-production additional item 1
      OUT     M7827  ; Non-production additional item 1
      MPP
      ANI     M7827  ; Non-production additional item 1
      MPS
      AND     M7924  ; Non-production additional item 2
      OUT     M7828  ; Non-production additional item 2
      MPP
      ANI     M7828  ; Non-production additional item 2
      OUT     M7799  ; Production time
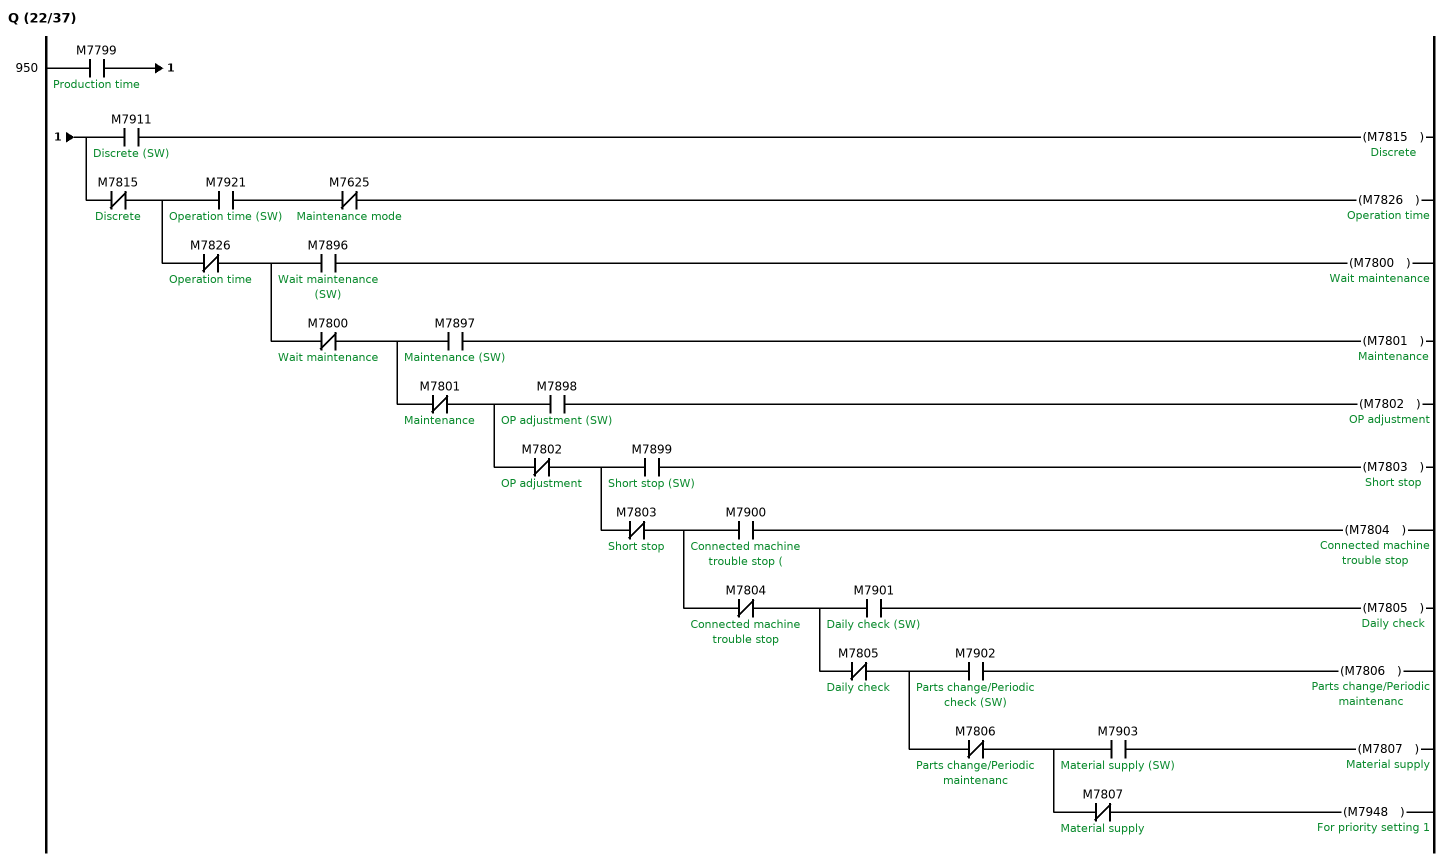
950   LD      M7799  ; Production time
      MPS
      AND     M7911  ; Discrete (SW)
      OUT     M7815  ; Discrete
      MPP
      ANI     M7815  ; Discrete
      MPS
      AND     M7921  ; Operation time (SW)
      ANI     M7625  ; Maintenance mode
      OUT     M7826  ; Operation time
      MPP
      ANI     M7826  ; Operation time
      MPS
      AND     M7896  ; Wait maintenance (SW)
      OUT     M7800  ; Wait maintenance
      MPP
      ANI     M7800  ; Wait maintenance
      MPS
      AND     M7897  ; Maintenance (SW)
      OUT     M7801  ; Maintenance
      MPP
      ANI     M7801  ; Maintenance
      MPS
      AND     M7898  ; OP adjustment (SW)
      OUT     M7802  ; OP adjustment
      MPP
      ANI     M7802  ; OP adjustment
      MPS
      AND     M7899  ; Short stop (SW)
      OUT     M7803  ; Short stop
      MPP
      ANI     M7803  ; Short stop
      MPS
      AND     M7900  ; Connected machine trouble stop (
      OUT     M7804  ; Connected machine trouble stop
      MPP
      ANI     M7804  ; Connected machine trouble stop
      MPS
      AND     M7901  ; Daily check (SW)
      OUT     M7805  ; Daily check
      MPP
      ANI     M7805  ; Daily check
      MPS
      AND     M7902  ; Parts change/Periodic check (SW)
      OUT     M7806  ; Parts change/Periodic maintenanc
      MPP
      ANI     M7806  ; Parts change/Periodic maintenanc
      MPS
      AND     M7903  ; Material supply (SW)
      OUT     M7807  ; Material supply
      MPP
      ANI     M7807  ; Material supply
      OUT     M7948  ; For priority setting 1
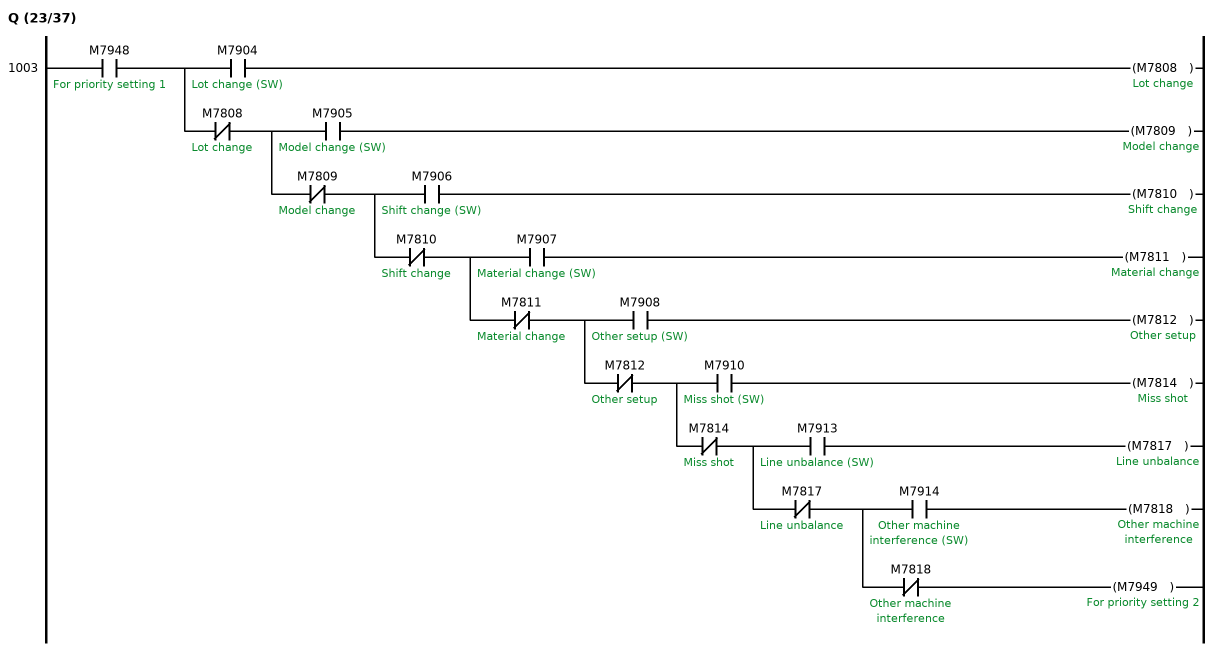
1003  LD      M7948  ; For priority setting 1
      MPS
      AND     M7904  ; Lot change (SW)
      OUT     M7808  ; Lot change
      MPP
      ANI     M7808  ; Lot change
      MPS
      AND     M7905  ; Model change (SW)
      OUT     M7809  ; Model change
      MPP
      ANI     M7809  ; Model change
      MPS
      AND     M7906  ; Shift change (SW)
      OUT     M7810  ; Shift change
      MPP
      ANI     M7810  ; Shift change
      MPS
      AND     M7907  ; Material change (SW)
      OUT     M7811  ; Material change
      MPP
      ANI     M7811  ; Material change
      MPS
      AND     M7908  ; Other setup (SW)
      OUT     M7812  ; Other setup
      MPP
      ANI     M7812  ; Other setup
      MPS
      AND     M7910  ; Miss shot (SW)
      OUT     M7814  ; Miss shot
      MPP
      ANI     M7814  ; Miss shot
      MPS
      AND     M7913  ; Line unbalance (SW)
      OUT     M7817  ; Line unbalance
      MPP
      ANI     M7817  ; Line unbalance
      MPS
      AND     M7914  ; Other machine interference (SW)
      OUT     M7818  ; Other machine interference
      MPP
      ANI     M7818  ; Other machine interference
      OUT     M7949  ; For priority setting 2
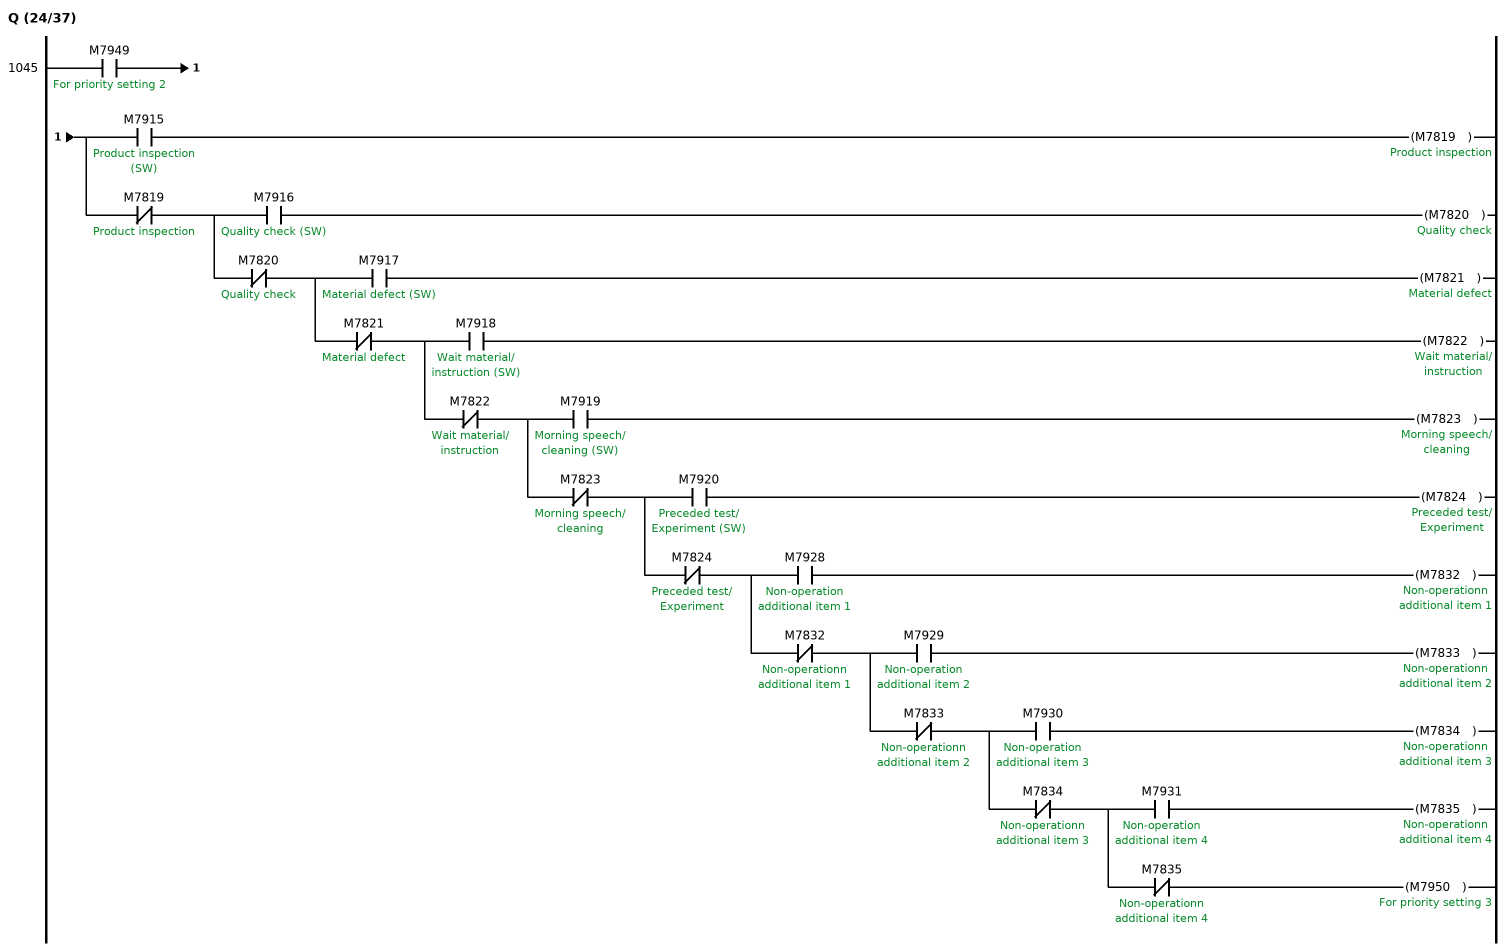
1045  LD      M7949  ; For priority setting 2
      MPS
      AND     M7915  ; Product inspection (SW)
      OUT     M7819  ; Product inspection
      MPP
      ANI     M7819  ; Product inspection
      MPS
      AND     M7916  ; Quality check (SW)
      OUT     M7820  ; Quality check
      MPP
      ANI     M7820  ; Quality check
      MPS
      AND     M7917  ; Material defect (SW)
      OUT     M7821  ; Material defect
      MPP
      ANI     M7821  ; Material defect
      MPS
      AND     M7918  ; Wait material/instruction (SW)
      OUT     M7822  ; Wait material/instruction
      MPP
      ANI     M7822  ; Wait material/instruction
      MPS
      AND     M7919  ; Morning speech/cleaning (SW)
      OUT     M7823  ; Morning speech/cleaning
      MPP
      ANI     M7823  ; Morning speech/cleaning
      MPS
      AND     M7920  ; Preceded test/Experiment (SW)
      OUT     M7824  ; Preceded test/Experiment
      MPP
      ANI     M7824  ; Preceded test/Experiment
      MPS
      AND     M7928  ; Non-operation additional item 1
      OUT     M7832  ; Non-operationn additional item 1
      MPP
      ANI     M7832  ; Non-operationn additional item 1
      MPS
      AND     M7929  ; Non-operation additional item 2
      OUT     M7833  ; Non-operationn additional item 2
      MPP
      ANI     M7833  ; Non-operationn additional item 2
      MPS
      AND     M7930  ; Non-operation additional item 3
      OUT     M7834  ; Non-operationn additional item 3
      MPP
      ANI     M7834  ; Non-operationn additional item 3
      MPS
      AND     M7931  ; Non-operation additional item 4
      OUT     M7835  ; Non-operationn additional item 4
      MPP
      ANI     M7835  ; Non-operationn additional item 4
      OUT     M7950  ; For priority setting 3
